FUNCTION F_AmphosMRC_Error : FB_AmphosMRC
VAR_INPUT
END_VAR
VAR
	fbAmphosMRC : FB_AmphosMRC;
END_VAR

fbAmphosMRC(
	bAmphosOn := TRUE,
	bMRC := FALSE
);
F_AmphosMRC_Error := fbAmphosMRC;

END_FUNCTION

(* stored: Version 1.1.0.1, ProductVersion 3.1.4020.14
   POU F_AmphosMRC_Error: Id {9bd8c8e0-99f9-4360-8a25-2ba957d3b608}, SpecialFunc None *)
